TYPE ST_Proportionair :
STRUCT
	
(* Control *)
xEnable	:	BOOL;
iSetpoint	:	INT;
iSetpointRaw	:	INT;
iHiLimit	:	INT;
iLoLimit	:	INT;

(* Readback *)
xStable	:	BOOL;//TTL signal from the proportionair controller that the pressure is stable
iPressure	:	INT;
iPressureRaw : INT;


END_STRUCT
END_TYPE

(* stored: Version 1.1.0.1, ProductVersion 3.1.0.26
   DUT ST_Proportionair: Id {1cb50253-0c45-4afc-8e14-284b1dbf64b6} *)
